// TIA Portal project "Sortiranje kutija" (V17)

(* hardware
DEVICE "S71500/ET200MP-Station_1"  S7-1500 station
   slot 0: "Profilschiene_0"  6ES7 590-1***0-0AA0
   slot 1: "PLC_1"  CPU 1511-1 PN  6ES7 511-1AK00-0AB0  V1.8
   slot 2: "AI 8xU/I/RTD/TC ST_1"  AI 8xU/I/RTD/TC ST  6ES7 531-7KF00-0AB0  V2.0
   slot 3: "AI 8xU/I/RTD/TC ST_2"  AI 8xU/I/RTD/TC ST  6ES7 531-7KF00-0AB0  V2.0
   slot 4: "AI 8xU/I/RTD/TC ST_3"  AI 8xU/I/RTD/TC ST  6ES7 531-7KF00-0AB0  V2.0
   slot 5: "AI 8xU/I/RTD/TC ST_4"  AI 8xU/I/RTD/TC ST  6ES7 531-7KF00-0AB0  V2.0
   slot 6: "DI 16x24VDC BA_1"  DI 16x24VDC BA  6ES7 521-1BH10-0AA0  V1.0
*)

// ===== PLC "PLC_1"  CPU 1511-1 PN =====

VAR_GLOBAL   // PLC tag table "Standard-Variablentabelle"
   "High_sensor" AT %E0.0 : Bool;
   "Low_sensor" AT %E0.1 : Bool;
   "Pallet_sensor" AT %I0.2 : Bool;
   "Loaded" AT %I0.3 : Bool;
   "Left_entry" AT %I0.4 : Bool;
   "Left_exit" AT %I0.5 : Bool;
   "Right_entry" AT %I0.6 : Bool;
   "Right_exit" AT %I0.7 : Bool;
   "Start" AT %I1.0 : Bool;
   "Reset" AT %I1.1 : Bool;
   "Stop" AT %I1.2 : Bool;
   "Emergency_stop" AT %I1.3 : Bool;
   "Auto" AT %I1.4 : Bool;
   "Factory_IO" AT %I1.5 : Bool;
   "Conveyor_entry" AT %Q0.0 : Bool;
   "Load" AT %Q0.1 : Bool;
   "Unload" AT %Q0.2 : Bool;
   "Trans_left" AT %Q0.3 : Bool;
   "Trans_right" AT %Q0.4 : Bool;
   "Conveyor_left" AT %Q0.5 : Bool;
   "Conveyor_right" AT %Q0.6 : Bool;
   "Start_light" AT %Q0.7 : Bool;
   "Reset_light" AT %Q1.0 : Bool;
   "Stop_light" AT %Q1.1 : Bool;
   "Counter" AT %QW30 : Int;
   "Tag_1" AT %M0.0 : Bool;
   "low_sensor_pom" AT %M0.1 : Bool;
   "Tag_3" AT %M0.2 : Bool;
   "High_sensor_pom" AT %M0.3 : Bool;
   "Tag_5" AT %M0.4 : Bool;
   "loaded_pom" AT %M0.5 : Bool;
   "Tag_7" AT %M0.6 : Bool;
   "Tag_8" AT %M0.7 : Bool;
   "Tag_9" AT %M2.0 : Bool;
   "left_entry_poz" AT %M2.1 : Bool;
   "Tag_11" AT %M2.2 : Bool;
   "right_entry_poz" AT %M2.3 : Bool;
   "Tag_13" AT %M2.4 : Bool;
   "left_entry_neg" AT %M2.5 : Bool;
   "Tag_15" AT %M2.6 : Bool;
   "right_entry_neg" AT %M2.7 : Bool;
   "Tag_17" AT %M3.0 : Bool;
   "left_exit_pom" AT %M3.1 : Bool;
   "right_exit_pom" AT %M3.2 : Bool;
   "Tag_20" AT %M3.3 : Bool;
   "Tag_21" AT %M4.0 : Bool;
   "Tag_22" AT %M4.1 : Bool;
END_VAR

// folder: System blocks/Program resources

DATA_BLOCK "IEC_Timer_0_DB"   // DB1
{ S7_Optimized_Access := 'TRUE' }
AUTHOR : Simatic
FAMILY : IEC
NAME : IEC_TMR
VERSION : 1.0
// stored: InstanceOfName IEC_TIMER
"IEC_TIMER"
BEGIN
END_DATA_BLOCK

DATA_BLOCK "IEC_Timer_0_DB_1"   // DB2
{ S7_Optimized_Access := 'TRUE' }
AUTHOR : Simatic
FAMILY : IEC
NAME : IEC_TMR
VERSION : 1.0
// stored: InstanceOfName IEC_TIMER
"IEC_TIMER"
BEGIN
END_DATA_BLOCK

// folder: (top level)

FUNCTION "Block_1" : Void   // FC1, LAD
{ S7_Optimized_Access := 'TRUE' }
VERSION : 0.1
   VAR_TEMP   // added for the SCL form of the ladder/FBD networks
      _w1 : Bool;
   END_VAR
BEGIN

REGION Network 1
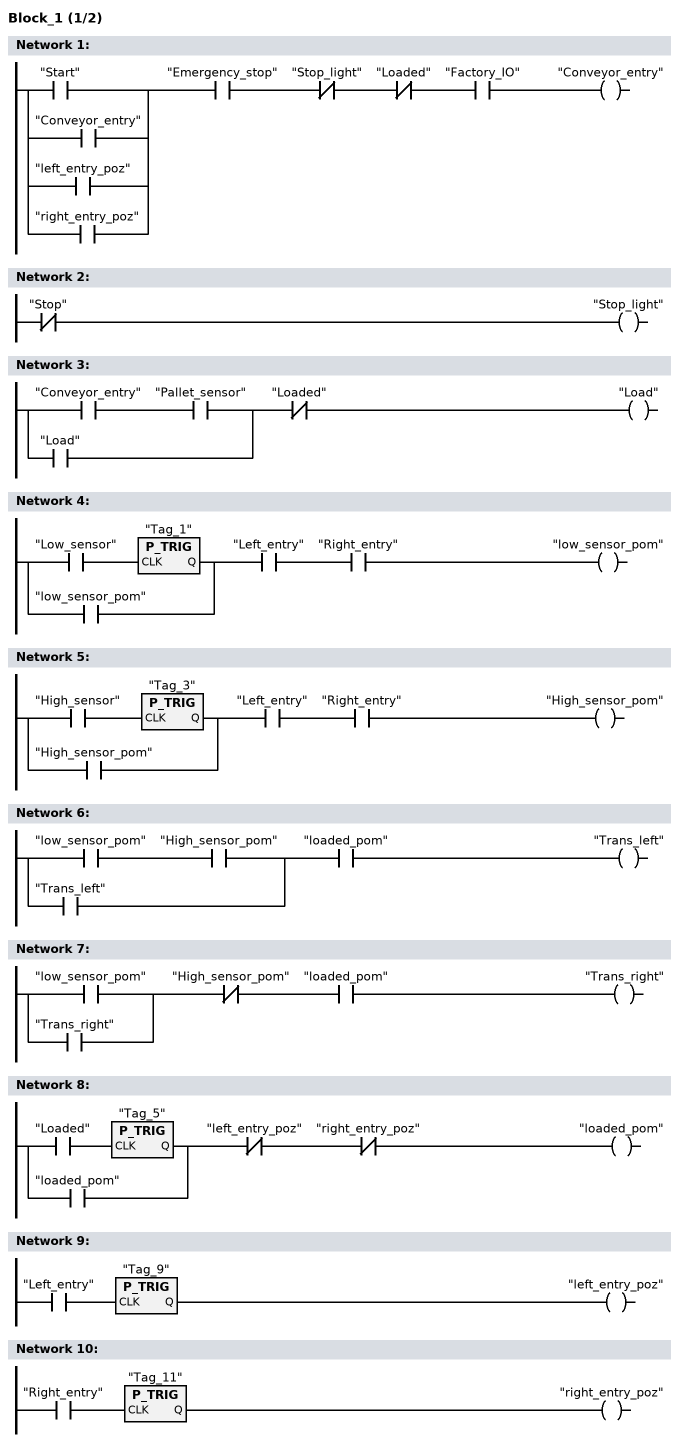
   RUNG wire#powerrail
      Contact( "Start" )
      wire#w1
      Contact( "Emergency_stop" )
      I_Contact( "Stop_light" )
      I_Contact( "Loaded" )
      Contact( "Factory_IO" )
      Coil( "Conveyor_entry" )
   END_RUNG
   RUNG wire#powerrail
      Contact( "Conveyor_entry" )
   END_RUNG wire#w1
   RUNG wire#powerrail
      Contact( "left_entry_poz" )
   END_RUNG wire#w1
   RUNG wire#powerrail
      Contact( "right_entry_poz" )
   END_RUNG wire#w1
   // the same network as SCL:
   "Conveyor_entry" := ("Start" OR "Conveyor_entry" OR "left_entry_poz" OR "right_entry_poz") AND "Emergency_stop" AND NOT "Stop_light" AND NOT "Loaded" AND "Factory_IO";
END_REGION

REGION Network 2
   RUNG wire#powerrail
      I_Contact( "Stop" )
      Coil( "Stop_light" )
   END_RUNG
   // the same network as SCL:
   "Stop_light" := NOT "Stop";
END_REGION

REGION Network 3
   RUNG wire#powerrail
      Contact( "Conveyor_entry" )
      Contact( "Pallet_sensor" )
      wire#w1
      I_Contact( "Loaded" )
      Coil( "Load" )
   END_RUNG
   RUNG wire#powerrail
      Contact( "Load" )
   END_RUNG wire#w1
   // the same network as SCL:
   "Load" := (("Conveyor_entry" AND "Pallet_sensor") OR "Load") AND NOT "Loaded";
END_REGION

REGION Network 4
   RUNG wire#powerrail
      Contact( "Low_sensor" )
      P_Trig( "Tag_1" )
      wire#w1
      Contact( "Left_entry" )
      Contact( "Right_entry" )
      Coil( "low_sensor_pom" )
   END_RUNG
   RUNG wire#powerrail
      Contact( "low_sensor_pom" )
   END_RUNG wire#w1
   // the same network as SCL:
   #_w1 := "Low_sensor" AND NOT "Tag_1";   // rising edge
   "Tag_1" := "Low_sensor";
   "low_sensor_pom" := (#_w1 OR "low_sensor_pom") AND "Left_entry" AND "Right_entry";
END_REGION

REGION Network 5
   RUNG wire#powerrail
      Contact( "High_sensor" )
      P_Trig( "Tag_3" )
      wire#w1
      Contact( "Left_entry" )
      Contact( "Right_entry" )
      Coil( "High_sensor_pom" )
   END_RUNG
   RUNG wire#powerrail
      Contact( "High_sensor_pom" )
   END_RUNG wire#w1
   // the same network as SCL:
   #_w1 := "High_sensor" AND NOT "Tag_3";   // rising edge
   "Tag_3" := "High_sensor";
   "High_sensor_pom" := (#_w1 OR "High_sensor_pom") AND "Left_entry" AND "Right_entry";
END_REGION

REGION Network 6
   RUNG wire#powerrail
      Contact( "low_sensor_pom" )
      Contact( "High_sensor_pom" )
      wire#w1
      Contact( "loaded_pom" )
      Coil( "Trans_left" )
   END_RUNG
   RUNG wire#powerrail
      Contact( "Trans_left" )
   END_RUNG wire#w1
   // the same network as SCL:
   "Trans_left" := (("low_sensor_pom" AND "High_sensor_pom") OR "Trans_left") AND "loaded_pom";
END_REGION

REGION Network 7
   RUNG wire#powerrail
      Contact( "low_sensor_pom" )
      wire#w1
      I_Contact( "High_sensor_pom" )
      Contact( "loaded_pom" )
      Coil( "Trans_right" )
   END_RUNG
   RUNG wire#powerrail
      Contact( "Trans_right" )
   END_RUNG wire#w1
   // the same network as SCL:
   "Trans_right" := ("low_sensor_pom" OR "Trans_right") AND NOT "High_sensor_pom" AND "loaded_pom";
END_REGION

REGION Network 8
   RUNG wire#powerrail
      Contact( "Loaded" )
      P_Trig( "Tag_5" )
      wire#w1
      I_Contact( "left_entry_poz" )
      I_Contact( "right_entry_poz" )
      Coil( "loaded_pom" )
   END_RUNG
   RUNG wire#powerrail
      Contact( "loaded_pom" )
   END_RUNG wire#w1
   // the same network as SCL:
   #_w1 := "Loaded" AND NOT "Tag_5";   // rising edge
   "Tag_5" := "Loaded";
   "loaded_pom" := (#_w1 OR "loaded_pom") AND NOT "left_entry_poz" AND NOT "right_entry_poz";
END_REGION

REGION Network 9
   RUNG wire#powerrail
      Contact( "Left_entry" )
      P_Trig( "Tag_9" )
      Coil( "left_entry_poz" )
   END_RUNG
   // the same network as SCL:
   #_w1 := "Left_entry" AND NOT "Tag_9";   // rising edge
   "Tag_9" := "Left_entry";
   "left_entry_poz" := #_w1;
END_REGION

REGION Network 10
   RUNG wire#powerrail
      Contact( "Right_entry" )
      P_Trig( "Tag_11" )
      Coil( "right_entry_poz" )
   END_RUNG
   // the same network as SCL:
   #_w1 := "Right_entry" AND NOT "Tag_11";   // rising edge
   "Tag_11" := "Right_entry";
   "right_entry_poz" := #_w1;
END_REGION

REGION Network 11
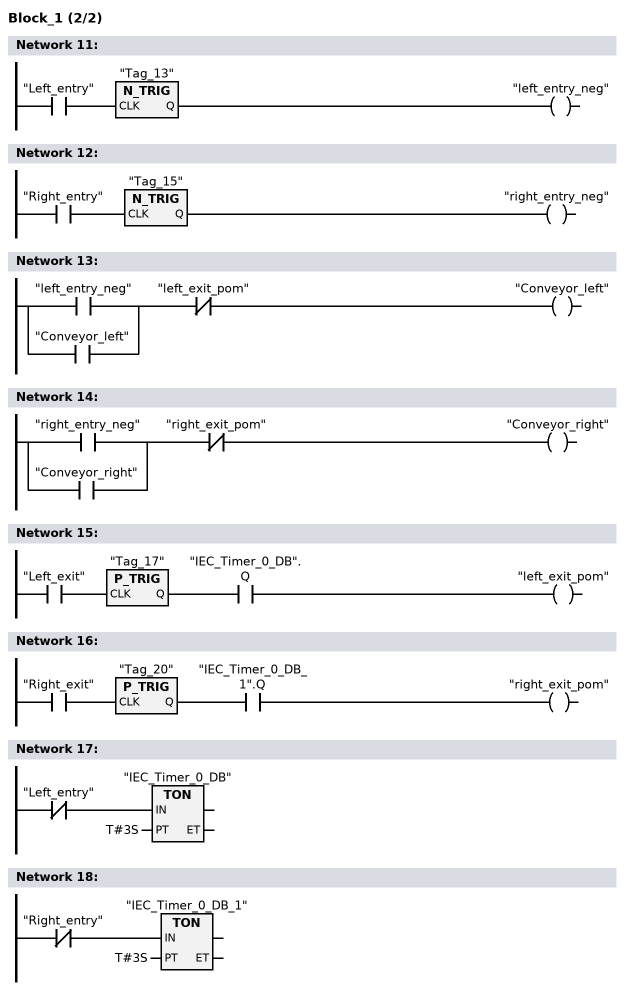
   RUNG wire#powerrail
      Contact( "Left_entry" )
      N_Trig( "Tag_13" )
      Coil( "left_entry_neg" )
   END_RUNG
   // the same network as SCL:
   #_w1 := NOT "Left_entry" AND "Tag_13";   // falling edge
   "Tag_13" := "Left_entry";
   "left_entry_neg" := #_w1;
END_REGION

REGION Network 12
   RUNG wire#powerrail
      Contact( "Right_entry" )
      N_Trig( "Tag_15" )
      Coil( "right_entry_neg" )
   END_RUNG
   // the same network as SCL:
   #_w1 := NOT "Right_entry" AND "Tag_15";   // falling edge
   "Tag_15" := "Right_entry";
   "right_entry_neg" := #_w1;
END_REGION

REGION Network 13
   RUNG wire#powerrail
      Contact( "left_entry_neg" )
      wire#w1
      I_Contact( "left_exit_pom" )
      Coil( "Conveyor_left" )
   END_RUNG
   RUNG wire#powerrail
      Contact( "Conveyor_left" )
   END_RUNG wire#w1
   // the same network as SCL:
   "Conveyor_left" := ("left_entry_neg" OR "Conveyor_left") AND NOT "left_exit_pom";
END_REGION

REGION Network 14
   RUNG wire#powerrail
      Contact( "right_entry_neg" )
      wire#w1
      I_Contact( "right_exit_pom" )
      Coil( "Conveyor_right" )
   END_RUNG
   RUNG wire#powerrail
      Contact( "Conveyor_right" )
   END_RUNG wire#w1
   // the same network as SCL:
   "Conveyor_right" := ("right_entry_neg" OR "Conveyor_right") AND NOT "right_exit_pom";
END_REGION

REGION Network 15
   RUNG wire#powerrail
      Contact( "Left_exit" )
      P_Trig( "Tag_17" )
      Contact( "IEC_Timer_0_DB".Q )
      Coil( "left_exit_pom" )
   END_RUNG
   // the same network as SCL:
   #_w1 := "Left_exit" AND NOT "Tag_17";   // rising edge
   "Tag_17" := "Left_exit";
   "left_exit_pom" := #_w1 AND "IEC_Timer_0_DB".Q;
END_REGION

REGION Network 16
   RUNG wire#powerrail
      Contact( "Right_exit" )
      P_Trig( "Tag_20" )
      Contact( "IEC_Timer_0_DB_1".Q )
      Coil( "right_exit_pom" )
   END_RUNG
   // the same network as SCL:
   #_w1 := "Right_exit" AND NOT "Tag_20";   // rising edge
   "Tag_20" := "Right_exit";
   "right_exit_pom" := #_w1 AND "IEC_Timer_0_DB_1".Q;
END_REGION

REGION Network 17
   "IEC_Timer_0_DB".TON(IN := NOT "Left_entry", PT := T#3S);
END_REGION

REGION Network 18
   "IEC_Timer_0_DB_1".TON(IN := NOT "Right_entry", PT := T#3S);
END_REGION
END_FUNCTION

FUNCTION "Block_2" : Void   // FC2, LAD
{ S7_Optimized_Access := 'TRUE' }
VERSION : 0.1
BEGIN
END_FUNCTION

FUNCTION "MHJ-PLC-Lab-Function-S71500" : Void   // FC9000, SCL
{ S7_Optimized_Access := 'TRUE' }
VERSION : 0.1
   VAR_TEMP
      Value : Byte;
      ForCounter : Int;
   END_VAR
   VAR CONSTANT
      Value_01_DW : DWord := 16#1223_5486;
      Value_02_DW : DWord := 16#A6C9_D1F5;
   END_VAR
BEGIN

   #Value:=PEEK(area := 16#82,
        dbNumber := 0,
        byteOffset := 511);
   #Value := #Value + 1;

   POKE(area := 16#82,
        dbNumber := 0,
        byteOffset := 511,
        value := #Value);

   POKE(area := 16#82,
        dbNumber := 0,
        byteOffset := 1016,
        value := #Value_01_DW);
   POKE(area := 16#82,
        dbNumber := 0,
        byteOffset := 1020,
        value := #Value_02_DW);

   FOR #ForCounter := 0 TO 63 DO
       #Value:=PEEK(area := 16#1,
            dbNumber := 0,
            byteOffset := #ForCounter);
       POKE(area := 16#81,
            dbNumber := 0,
            byteOffset := #ForCounter,
            value := #Value);
   END_FOR;
   #Value := PEEK(area := 16#1,
                  dbNumber := 0,
                  byteOffset := 512);
   POKE(area := 16#82,
        dbNumber := 0,
        byteOffset := 512,
        value := #Value);
END_FUNCTION

ORGANIZATION_BLOCK "Main"   // OB1, FBD, ProgramCycle
TITLE = "Main Program Sweep (Cycle)"
{ S7_Optimized_Access := 'TRUE' }
VERSION : 0.1
   VAR_INPUT
      Initial_Call : Bool;   // Initial call of this OB
      Remanence : Bool;   // =True, if remanent data are available
   END_VAR
BEGIN

REGION Network 1
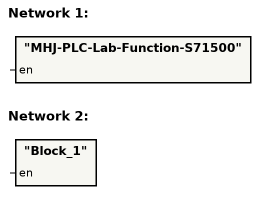
   "MHJ-PLC-Lab-Function-S71500"();
END_REGION

REGION Network 2
   "Block_1"();
END_REGION
END_ORGANIZATION_BLOCK